FUNCTION_BLOCK FB_LowTemperatureHeatingNetwork
VAR_INPUT
	stAmbientState : ST_AmbientState;
	
	//control struct for hnlt
	stHNLTControl : ST_LowTemperatureHeatingNetworkControl;	
END_VAR
VAR_OUTPUT
	//temperatures in buffer storage
	fTemperatureBufferStorage : REAL;
END_VAR
VAR
	//systems
	BufferStorage : FB_BufferStorage;
	OuterCapillaryTubeMats : FB_OuterCapillaryTubeMats;
	HVFASystem : FB_HVFAStorageSystem;
	
	//internal variables
	fSetPoint_HVFASystem : REAL;
END_VAR

//buffer storage system
BufferStorage();
fTemperatureBufferStorage := BufferStorage.fMidTemperature;

//producer

//consumer
OuterCapillaryTubeMats(bSetStatusOnAutomatic := stHNLTControl.bSetStatusOn_OuterCapillaryTubeMats,
	bAlgorithmPermission := stHNLTControl.bAlgorithmPermission,
	fSetPointAutomatic := stHNLTControl.fTargetTemperature,
	stAmbientState := stAmbientState);
	
//external storages
//setpoint depends on loading mode -> storage must be warmer than setpoint temperature in network
IF stHNLTControl.bLoading_HVFASystem THEN
	fSetPoint_HVFASystem := stHNLTControl.fTargetTemperature+5;
ELSE
	fSetPoint_HVFASystem := stHNLTControl.fTargetTemperature;
END_IF
HVFASystem(bSetStatusOnAutomatic := stHNLTControl.bSetStatusOn_HVFASystem,
	bAlgorithmPermission := stHNLTControl.bAlgorithmPermission,
	fSetPointAutomatic := fSetpoint_HVFASystem,
	bLoadingAutomatic := stHNLTControl.bLoading_HVFASystem);

END_FUNCTION_BLOCK

(* stored: Version 1.1.0.1, ProductVersion 3.1.4024.10
   POU FB_LowTemperatureHeatingNetwork: Id {41e3edb3-66e7-411c-a35e-b44e9a5d66f1}, SpecialFunc None *)
